# EPICS autosave request: xx_auto_icbTca_settings.req
$(P)$(T)POLARITY
$(P)$(T)THRESHOLD
$(P)$(T)SCA_ENABLE
$(P)$(T)READBACK.SCAN
$(P)$(T)PUR_ENABLE
$(P)$(T)PUR_AMP
$(P)$(T)TCA_SELECT
$(P)$(T)SCA1_GATE
$(P)$(T)SCA1_PUR
$(P)$(T)SCA1_LOW
$(P)$(T)SCA1_HI
$(P)$(T)SCA2_GATE
$(P)$(T)SCA2_PUR
$(P)$(T)SCA2_LOW
$(P)$(T)SCA2_HI
$(P)$(T)SCA3_GATE
$(P)$(T)SCA3_PUR
$(P)$(T)SCA3_LOW
$(P)$(T)SCA3_HI
$(P)$(T)ROI_SCA_ENABLE
$(P)$(T)SCA_CAL
